GLOBALCONSTANTS SubStrings (* Global constants *)
  (* Standard: 61499-1 *)
  (* Version 1.0, 2026-08-30, Franz Höpfinger, Meisterschulen am Ostbahnhof *)
  PACKAGE Meins::InputOutputTester::Button_AI_OPC_UA;
  VAR_GLOBAL CONSTANT
    AI_I1_RAW_WRITE : WSTRING := "opc_ua[WRITE;/Objects/Analog/I1/RAW,1:s=AI_I1_RAW]";
    AI_I1_PERCENT_WRITE : WSTRING := "opc_ua[WRITE;/Objects/Analog/I1/PERCENT,1:s=AI_I1_PERCENT]";
    AI_I2_RAW_WRITE : WSTRING := "opc_ua[WRITE;/Objects/Analog/I2/RAW,1:s=AI_I2_RAW]";
    AI_I2_PERCENT_WRITE : WSTRING := "opc_ua[WRITE;/Objects/Analog/I2/PERCENT,1:s=AI_I2_PERCENT]";
    AI_I3_RAW_WRITE : WSTRING := "opc_ua[WRITE;/Objects/Analog/I3/RAW,1:s=AI_I3_RAW]";
    AI_I3_PERCENT_WRITE : WSTRING := "opc_ua[WRITE;/Objects/Analog/I3/PERCENT,1:s=AI_I3_PERCENT]";
    AI_I4_RAW_WRITE : WSTRING := "opc_ua[WRITE;/Objects/Analog/I4/RAW,1:s=AI_I4_RAW]";
    AI_I4_PERCENT_WRITE : WSTRING := "opc_ua[WRITE;/Objects/Analog/I4/PERCENT,1:s=AI_I4_PERCENT]";
    AI_I5_RAW_WRITE : WSTRING := "opc_ua[WRITE;/Objects/Analog/I5/RAW,1:s=AI_I5_RAW]";
    AI_I5_PERCENT_WRITE : WSTRING := "opc_ua[WRITE;/Objects/Analog/I5/PERCENT,1:s=AI_I5_PERCENT]";
    AI_I6_RAW_WRITE : WSTRING := "opc_ua[WRITE;/Objects/Analog/I6/RAW,1:s=AI_I6_RAW]";
    AI_I6_PERCENT_WRITE : WSTRING := "opc_ua[WRITE;/Objects/Analog/I6/PERCENT,1:s=AI_I6_PERCENT]";
    AI_I7_RAW_WRITE : WSTRING := "opc_ua[WRITE;/Objects/Analog/I7/RAW,1:s=AI_I7_RAW]";
    AI_I7_PERCENT_WRITE : WSTRING := "opc_ua[WRITE;/Objects/Analog/I7/PERCENT,1:s=AI_I7_PERCENT]";
    AI_I8_RAW_WRITE : WSTRING := "opc_ua[WRITE;/Objects/Analog/I8/RAW,1:s=AI_I8_RAW]";
    AI_I8_PERCENT_WRITE : WSTRING := "opc_ua[WRITE;/Objects/Analog/I8/PERCENT,1:s=AI_I8_PERCENT]";
    Q01_READ : WSTRING := "opc_ua[READ;/Objects/DigitalOutput/Q01,1:s=Q01]";
    Q01_WRITE : WSTRING := "opc_ua[WRITE;/Objects/DigitalOutput/Q01,1:s=Q01]";
    Q02_READ : WSTRING := "opc_ua[READ;/Objects/DigitalOutput/Q02,1:s=Q02]";
    Q02_WRITE : WSTRING := "opc_ua[WRITE;/Objects/DigitalOutput/Q02,1:s=Q02]";
    Q03_READ : WSTRING := "opc_ua[READ;/Objects/DigitalOutput/Q03,1:s=Q03]";
    Q03_WRITE : WSTRING := "opc_ua[WRITE;/Objects/DigitalOutput/Q03,1:s=Q03]";
    Q04_READ : WSTRING := "opc_ua[READ;/Objects/DigitalOutput/Q04,1:s=Q04]";
    Q04_WRITE : WSTRING := "opc_ua[WRITE;/Objects/DigitalOutput/Q04,1:s=Q04]";
    Q05_READ : WSTRING := "opc_ua[READ;/Objects/DigitalOutput/Q05,1:s=Q05]";
    Q05_WRITE : WSTRING := "opc_ua[WRITE;/Objects/DigitalOutput/Q05,1:s=Q05]";
    Q06_READ : WSTRING := "opc_ua[READ;/Objects/DigitalOutput/Q06,1:s=Q06]";
    Q06_WRITE : WSTRING := "opc_ua[WRITE;/Objects/DigitalOutput/Q06,1:s=Q06]";
    Q07_READ : WSTRING := "opc_ua[READ;/Objects/DigitalOutput/Q07,1:s=Q07]";
    Q07_WRITE : WSTRING := "opc_ua[WRITE;/Objects/DigitalOutput/Q07,1:s=Q07]";
    Q08_READ : WSTRING := "opc_ua[READ;/Objects/DigitalOutput/Q08,1:s=Q08]";
    Q08_WRITE : WSTRING := "opc_ua[WRITE;/Objects/DigitalOutput/Q08,1:s=Q08]";
    Q09_READ : WSTRING := "opc_ua[READ;/Objects/DigitalOutput/Q09,1:s=Q09]";
    Q09_WRITE : WSTRING := "opc_ua[WRITE;/Objects/DigitalOutput/Q09,1:s=Q09]";
    Q10_READ : WSTRING := "opc_ua[READ;/Objects/DigitalOutput/Q10,1:s=Q10]";
    Q10_WRITE : WSTRING := "opc_ua[WRITE;/Objects/DigitalOutput/Q10,1:s=Q10]";
    Q11_READ : WSTRING := "opc_ua[READ;/Objects/DigitalOutput/Q11,1:s=Q11]";
    Q11_WRITE : WSTRING := "opc_ua[WRITE;/Objects/DigitalOutput/Q11,1:s=Q11]";
    Q12_READ : WSTRING := "opc_ua[READ;/Objects/DigitalOutput/Q12,1:s=Q12]";
    Q12_WRITE : WSTRING := "opc_ua[WRITE;/Objects/DigitalOutput/Q12,1:s=Q12]";
    Tick_WRITE : WSTRING := "opc_ua[WRITE;/Objects/System/Tick,1:s=System.Tick]";
  END_VAR
END_GLOBALCONSTANTS
